FUNCTION_BLOCK ZONE_VIEW (* Data Presentation for an HVAC Zone *)
  (* Standard: 61499-1; Classification: HMI; ApplicationDomain: HVAC; Function: View; Type: Zone; Description: HVAC Zone View *)
  (* Version 0.0, 2006-04-06, JHC, Holobloc Inc *)
  (* Compiler header: package fb.rt.hvac; *)
  (* Compiler Java Sun JDK 1.5.0 *)
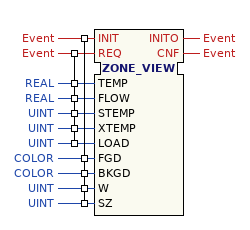
  EVENT_INPUT
    INIT WITH W, SZ, FGD, BKGD; (* Initialization *)
    REQ WITH TEMP, XTEMP, LOAD, STEMP, FLOW; (* Data Display Request *)
  END_EVENT
  EVENT_OUTPUT
    INITO; (* INIT Confirmation *)
    CNF; (* REQ Confirmation *)
  END_EVENT
  VAR_INPUT
    TEMP : REAL; (* Room Temperature, deg. F *)
    FLOW : REAL; (* Air Flow, CFM *)
    STEMP : UINT; (* Supply Air Temperature, deg F *)
    XTEMP : UINT; (* Exterior Temperature, deg F *)
    LOAD : UINT; (* Heat Load, KBTU/hr *)
    FGD : COLOR := COLOR#white; (* Foreground Color *)
    BKGD : COLOR := COLOR#blue; (* Background Color *)
    W : UINT; (* Square room side dimension in pixels *)
    SZ : UINT := 12; (* Font size in points *)
  END_VAR
  SERVICE APPLICATION/RESOURCE
    SEQUENCE initialize
      APPLICATION.INIT(FGD,BKGD,W,SZ) -> RESOURCE.initialize(FGD,BKGD,W,SZ) -> APPLICATION.INITO();
    END_SEQUENCE
    SEQUENCE request
      APPLICATION.REQ(TEMP,FLOW,STEMP,XTEMP,LOAD) -> RESOURCE.request(TEMP,FLOW,STEMP,XTEMP,LOAD) -> APPLICATION.CNF();
    END_SEQUENCE
  END_SERVICE
END_FUNCTION_BLOCK
